FUNCTION_BLOCK A2X_2X_TO_2AX (* Composite FB for convert A2X to 2 AX *)
  (* Standard: 61499-2; Description: Copyright (c) 2024 HR Agrartechnik GmbH This program and the accompanying materials are made available under the terms of the Eclipse Public License 2.0 which is available at https://www.eclipse.org/legal/epl-2.0/ SPDX-License-Identifier: EPL-2.0 *)
  (* Version 1.0, 2024-04-24, Franz Höpfinger, HR Agrartechnik GmbH *)
  PACKAGE adapter::conversion::unidirectional;
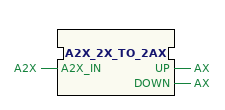
  SOCKETS
    A2X_IN : adapter::types::unidirectional::A2X; (* Adapter Input *)
  END_SOCKETS
  PLUGS
    UP : adapter::types::unidirectional::AX; (* TRUE = forward, up, right, clockwise *)
    DOWN : adapter::types::unidirectional::AX; (* TRUE = backward, down, left, counter-clockwise *)
  END_PLUGS
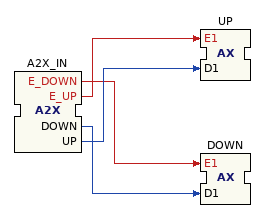
  EVENT_CONNECTIONS
    A2X_IN.E_DOWN TO DOWN.E1;
    A2X_IN.E_UP TO UP.E1;
  END_CONNECTIONS
  DATA_CONNECTIONS
    A2X_IN.DOWN TO DOWN.D1;
    A2X_IN.UP TO UP.D1;
  END_CONNECTIONS
END_FUNCTION_BLOCK
